TYPE EcCoeSdo_Input_typ :
	STRUCT
		Read	: EcCoeSdo_Par_Read_typ;
		Write	: EcCoeSdo_Par_Write_typ;
	END_STRUCT
END_TYPE

(* stored: Version 1.1.0.1, ProductVersion 3.1.4024.3
   DUT EcCoeSdo_Input_typ: Id {c45d2690-6888-06aa-1ba1-8a26e8e85ab2} *)
